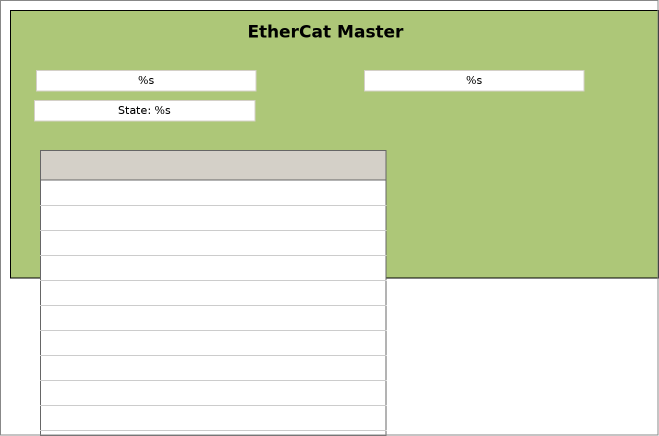
VISUALIZATION V_EtherCatMasterComponent  // 659x436
VAR_IN_OUT
	EtherCatMaster_HMI : ST_EtherCatMaster_HMI;
END_VAR
(*
		AmsNetID			: T_AMSNETID;
		CfgSlaveCount		: UINT;
		EcSlavesState		: ARRAY[0..EC_MAX_SLAVES] OF ST_EcSlaveState;
		ConfiguredSlaveInfo : ARRAY[0..EC_MAX_SLAVES] OF ST_EcSlaveConfigData;
		EcSlaveTopologyInfo : ARRAY[0..EC_MAX_SLAVES] OF ST_TopologyDataEx;
*)
    RoundedRectangle (10,10 649x268)
    Label (41,13 569x37), "EtherCat Master"
    Textfield (34,100 221x21), "State: %s", text variable: HMI.Status.State
    Textfield (36,70 220x21), "%s", text variable: EtherCatMaster_HMI.Status.
    Table (40,150 346x286)
    Textfield (364,70 220x21), "%s", text variable: EtherCatMaster_HMI.Status.ConfiguredSlaveInfo
END_VISUALIZATION

(* stored: Version 1.1.0.1, ProductVersion 3.1.4024.15
   Visu V_EtherCatMasterComponent: Id {860cbfe9-f36c-4950-ba62-ea1feb660ec2} *)
